FUNCTION_BLOCK TwoStateInd (* Composite Function Block Type *)
  (* Standard: 61499-2 *)
  (* Version 0.2, 2003-12-05, JHC, Rockwell Automation, Renamed from NEWCOMPFB. *)
  (* Version 0.1, 2002-01-08, JHC, Rockwell Automation, Added DLY FB as example. *)
  (* Version 0.0, 2000-05-27, JHC, Rockwell Automation *)
  (* Compiler header: package fb.rt.template; *)
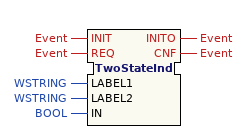
  EVENT_INPUT
    INIT; (* Initialization Request *)
    REQ; (* Normal Execution Request *)
  END_EVENT
  EVENT_OUTPUT
    INITO; (* Initialization Confirm *)
    CNF; (* Execution Confirmation *)
  END_EVENT
  VAR_INPUT
    LABEL1 : WSTRING;
    LABEL2 : WSTRING;
    IN : BOOL;
  END_VAR
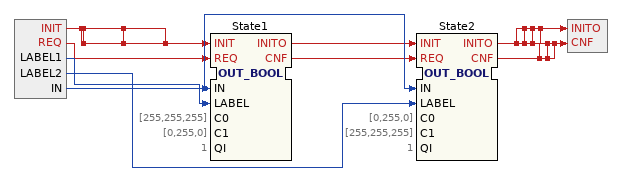
  FBS
    State1 : OUT_BOOL(C0 := [255,255,255], C1 := [0,255,0], QI := 1);
    State2 : OUT_BOOL(C0 := [0,255,0], C1 := [255,255,255], QI := 1);
  END_FBS
  EVENT_CONNECTIONS
    INIT TO State1.INIT;
    State1.INITO TO State2.INIT;
    REQ TO State1.REQ;
    State1.CNF TO State2.REQ;
    State2.INITO TO INITO;
    State2.CNF TO CNF;
    INIT TO State1.INIT;
    State1.INITO TO State2.INIT;
    REQ TO State1.REQ;
    State1.CNF TO State2.REQ;
    State2.INITO TO INITO;
    State2.CNF TO CNF;
    INIT TO State1.INIT;
    State1.INITO TO State2.INIT;
    REQ TO State1.REQ;
    State1.CNF TO State2.REQ;
    State2.INITO TO INITO;
    State2.CNF TO CNF;
    INIT TO State1.INIT;
    State1.INITO TO State2.INIT;
    REQ TO State1.REQ;
    State1.CNF TO State2.REQ;
    State2.INITO TO INITO;
    State2.CNF TO CNF;
  END_CONNECTIONS
  DATA_CONNECTIONS
    IN TO State1.IN;
    IN TO State2.IN;
    LABEL1 TO State1.LABEL;
    LABEL2 TO State2.LABEL;
    IN TO State1.IN;
    IN TO State2.IN;
    LABEL1 TO State1.LABEL;
    LABEL2 TO State2.LABEL;
    IN TO State1.IN;
    IN TO State2.IN;
    LABEL1 TO State1.LABEL;
    LABEL2 TO State2.LABEL;
    IN TO State1.IN;
    IN TO State2.IN;
    LABEL1 TO State1.LABEL;
    LABEL2 TO State2.LABEL;
  END_CONNECTIONS
END_FUNCTION_BLOCK
